{attribute 'pack_mode' := '2'}
TYPE ST_INSTANCE_CTRL :
STRUCT
  Cmd     : E_INSTANCE_CMD;
END_STRUCT
END_TYPE

(* stored: Version 1.1.0.1, ProductVersion 3.1.4026.18
   DUT ST_INSTANCE_CTRL: Id {8fd044db-5f6b-4e20-b3ae-8230cfc86880} *)
